{attribute 'GeneratedUsingTerminal: AT2026-0250-0019'}
{attribute addProperty BoxType "AT2026-0250-0019"}
{attribute addProperty Id "A_0077_AT2001_5250_0018_AT2001_5250AT2001_01D6DEDF80"}
{attribute addProperty CRC "936959846"}
{attribute addProperty Size "80"}
TYPE A_0065_AT2026_0250_0019_AT2026_0250_37D8DF66 EXTENDS AT2026_86175B41 :
STRUCT
	{attribute addProperty Name "A_0077_AT2001_5250_0018_AT2001_5250"}
	A_0077_AT2001_5250_0018_AT2001_5250 : AT2001_01D6DEDF;
END_STRUCT
END_TYPE

(* stored: Version 1.2.0.0, ProductVersion 3.1.4024.9
   DUT A_0065_AT2026_0250_0019_AT2026_0250_37D8DF66: Id {07aa5b2c-c288-41e1-bb97-2d74705904c9} *)
